FUNCTION_BLOCK Equipo_Motor_ATV320
VAR_INPUT
	wStatus			:UINT;
	wRpm_var		:WORD; // rpm actuales leidas del variador
	iVelo			:REAL; // set velocidad en %
	iRpmNom			:INT;// rpm nominales leidas del variador
	bCmdMarcha		:BOOL;
	bReverse		:BOOL;
	bParada_Quick	:BOOL;//parada rapida 16#0002
	bParada_Normal	:BOOL;//parada normal 16#0007
	Interlock	:BOOL;	//Deve estar em TRUE para liberar o funcionamento da bomba
END_VAR
VAR_OUTPUT
	bEnMarcha:BOOL;
	bAlr:BOOL;
	wControl:UINT;
	wEstado:WORD;
	iVelOUT:UINT;
	iRPM_a_HMI:INT; //rpm para el HMI

END_VAR
VAR
	Aux_Status:DINT;
	bMarcha:BOOL;
	TempoFuncionando:UDINT;	//Tempo de funcionamento do motor
	Acionamentos	:UDINT;	//Quantidade de acionamentos do motor
	TON_Horimetro: TON;
	RTRIG_Funcionamento: R_TRIG;
	ResetContadores: BOOL;
END_VAR


(*cuenta horas de marcha parciales*)
(*cuenta horas de marcha totales*)

(***********************************************************************Tratamiento PDO*)
wEstado := wStatus;
iVelOUT:=REAL_TO_UINT(iRpmNom*iVelo/100);// convierte velocidad solicitada en % a rpm
iRPM_a_HMI:=WORD_TO_INT (wRpm_var);

Aux_Status:= DINT_TO_UINT(wStatus) AND 16#007F;


(*Secuencia Marcha*)
IF bCmdMarcha AND Interlock THEN
	IF (Aux_Status=16#0050 OR Aux_Status =16#0060 OR Aux_Status =16#0080) THEN
		wControl:=16#0006;	
	END_IF
	IF Aux_Status=16#0031  THEN
		wControl:=16#0007;	
	END_IF
	IF Aux_Status=16#0033  THEN
		IF bReverse THEN	
			wControl:=16#080F;
		ELSE	
			wControl:=16#000F;
		END_IF
	END_IF	
END_IF

(*Secuencia Parada*)
IF  (NOT bCmdMarcha OR NOT Interlock) AND Aux_Status=16#0037 THEN
	IF bParada_Quick THEN
		wControl:=16#0002;//quick	
		ELSE
		wControl:=16#0007;//normal
	END_IF
END_IF 

(*Deshabilita tension*)
IF  Aux_Status=16#0017 THEN
	wControl:=16#0000;
END_IF 

(*Aviso Falla*)
IF (Aux_Status=16#0008 OR Aux_Status=16#0028 OR Aux_Status=16#000F OR Aux_Status=16#0038 OR Aux_Status=16#002F OR Aux_Status=16#0018 ) THEN
	bAlr:=1;
	ELSE
	bAlr:=0;	
	END_IF
	
(*Reset Falla*)
(*Estado*)
IF (Aux_Status=16#0037) THEN
	bEnMarcha:=1;
	
ELSE
	bEnMarcha:=0;	
END_IF

//Motor rodando
TON_Horimetro(IN:= bEnMarcha AND NOT TON_Horimetro.Q, PT:=T#1M);
IF TON_Horimetro.Q THEN
	TempoFuncionando := TempoFuncionando + 1;
END_IF

//Quantidade de acionamentos
RTRIG_Funcionamento(CLK:=bEnMarcha);
IF RTRIG_Funcionamento.Q THEN
	Acionamentos := Acionamentos + 1;
END_IF

//Reset contadores
IF ResetContadores THEN
	Acionamentos		:= 0;
	TempoFuncionando	:= 0;
	ResetContadores		:= FALSE;
END_IF


(***********************************************************************Tratamiento SDO*)

END_FUNCTION_BLOCK

(* stored: Version 1.1.0.1, ProductVersion 3.1.4024.14
   POU Equipo_Motor_ATV320: Id {b80954b0-0d87-49a3-b865-4d98fda21dcd}, SpecialFunc None *)
